# B&R Automation Studio project SCR
Automation Studio 4.0.18.71 SP

## Logical view

Binary libraries used (declarations not repeated): operator, runtime, astime, AsIecCon

### Global.var - Global variables
```iecst
(********************************************************************
 * COPYRIGHT --
 ********************************************************************
 * File: Global.var
 * Author: Arkadiusz
 * Created: April 16, 2018
 ********************************************************************
 * Global variables of project test2
 ********************************************************************)
VAR
	zadajnik : USINT;
	output2 : USINT;
	output1 : USINT;
	input3 : USINT;
	input2 : USINT;
	input1 : USINT;
	subs2Value : USINT;
	subs1Value : USINT;
	valuesSetFlag : USINT := 0;
END_VAR
```


### Program Logical/NastawaPWM (ANSIC) - Program

#### NastawaPWMCyclic.c - Cyclic code
```c
/********************************************************************
 * COPYRIGHT --
 ********************************************************************
 * Program: NastawaPWM
 * File: NastawaPWMCyclic.c
 * Author: Arkadiusz
 * Created: April 23, 2018
 ********************************************************************
 * Implementation of program NastawaPWM
 ********************************************************************/

#include <bur/plctypes.h>

#ifdef _DEFAULT_INCLUDES
	#include <AsDefault.h>
#endif

void _CYCLIC NastawaPWMCyclic(void)
{
	const double mnoznik = 0.027;
	wynikNastawy = inputAnalogowy * mnoznik;

	inputPerc = wynikNastawy;
	inputT_Ms = 20000;
	const cycleTime = 10;
	cycleIterator = cycleIterator + 1;
	time = cycleIterator * cycleTime;
	upTime = ((double)inputPerc/100) * inputT_Ms;

	if (time < upTime)
	{
		out1 = 1;
	}
	else
	{
		out1 = 0;
	}

	if (time >= inputT_Ms)
	{
		time = 0;
		cycleIterator = 0;
	}
}
```

#### NastawaPWMInit.c - Initialization code
```c
/********************************************************************
 * COPYRIGHT --
 ********************************************************************
 * Program: NastawaPWM
 * File: NastawaPWMInit.c
 * Author: Arkadiusz
 * Created: April 23, 2018
 ********************************************************************
 * Implementation of program NastawaPWM
 ********************************************************************/

#include <bur/plctypes.h>

#ifdef _DEFAULT_INCLUDES
	#include <AsDefault.h>
#endif

void _INIT NastawaPWMInit(void)
{
	/* TODO: Add code here */
}
```

#### NastawaPWM.var - Local variables
```iecst
(********************************************************************
 * COPYRIGHT --
 ********************************************************************
 * Program: NastawaPWM
 * File: NastawaPWM.var
 * Author: Arkadiusz
 * Created: April 23, 2018
 ********************************************************************
 * Local variables of program NastawaPWM
 ********************************************************************)
VAR
	upTime : REAL;
	time : LREAL;
	inputPerc : USINT := 0;
	out1 : USINT := 0;
	cycleIterator : INT := 0;
	inputT_Ms : UDINT := 0;
	inputAnalogowy : INT;
	wynikNastawy : USINT;
	inputVolt : REAL;
END_VAR
```

### Program Logical/PWM (ANSIC) - Program

#### PWMCyclic.c - Cyclic code
```c
/********************************************************************
 * COPYRIGHT --
 ********************************************************************
 * Program: Testowy
 * File: TestowyCyclic.c
 * Author: Arkadiusz
 * Created: April 16, 2018
 ********************************************************************
 * Implementation of program Testowy
 ********************************************************************/

#include <bur/plctypes.h>

#ifdef _DEFAULT_INCLUDES
	#include <AsDefault.h>
#endif

void _CYCLIC TestowyCyclic(void)
{
	inputPerc = 50;
	inputT_Ms = 20000;
	const cycleTime = 10;
	cycleIterator = cycleIterator + 1;
	time = cycleIterator * cycleTime;
	upTime = ((double)inputPerc/100) * inputT_Ms;

	if (time < upTime)
	{
		out1 = 1;
	}
	else
	{
		out1 = 0;
	}

	if (time >= inputT_Ms)
	{
		time = 0;
		cycleIterator = 0;
	}

}
```

#### PWMInit.c - Initialization code
```c
/********************************************************************
 * COPYRIGHT --
 ********************************************************************
 * Program: Testowy
 * File: TestowyInit.c
 * Author: Arkadiusz
 * Created: April 16, 2018
 ********************************************************************
 * Implementation of program Testowy
 ********************************************************************/

#include <bur/plctypes.h>

#ifdef _DEFAULT_INCLUDES
	#include <AsDefault.h>
#endif

void _INIT TestowyInit(void)
{
	out1 = 0;

}
```

#### PWM.var - Local variables
```iecst
(********************************************************************
 * COPYRIGHT --
 ********************************************************************
 * Program: Testowy
 * File: Testowy.var
 * Author: Arkadiusz
 * Created: April 16, 2018
 ********************************************************************
 * Local variables of program Testowy
 ********************************************************************)
VAR
	upTime : REAL;
	time : LREAL;
	inputPerc : USINT := 0;
	out1 : USINT := 0;
	cycleIterator : INT := 0;
	inputT_Ms : UDINT := 0;
END_VAR
```

### Program Logical/Nastawa (ANSIC) - nastawaProgram

#### NastawaCyclic.c - Cyclic code
```c
/********************************************************************
 * COPYRIGHT --
 ********************************************************************
 * Program: Nastawa
 * File: NastawaCyclic.c
 * Author: Arkadiusz
 * Created: April 23, 2018
 ********************************************************************
 * Implementation of program Nastawa
 ********************************************************************/

#include <bur/plctypes.h>

#ifdef _DEFAULT_INCLUDES
	#include <AsDefault.h>
#endif

void _CYCLIC NastawaCyclic(void)
{
	const double mnoznik = 100.0/32768;
	wynikNastawy = (int) ( ( (double) inputAnalogowy ) * mnoznik);
	zadajnik = wynikNastawy;

}
```

#### NastawaInit.c - Initialization code
```c
/********************************************************************
 * COPYRIGHT --
 ********************************************************************
 * Program: Nastawa
 * File: NastawaInit.c
 * Author: Arkadiusz
 * Created: April 23, 2018
 ********************************************************************
 * Implementation of program Nastawa
 ********************************************************************/

#include <bur/plctypes.h>

#ifdef _DEFAULT_INCLUDES
	#include <AsDefault.h>
#endif

void _INIT NastawaInit(void)
{
	/* TODO: Add code here */
}
```

#### Nastawa.var - Local variables
```iecst
(********************************************************************
 * COPYRIGHT --
 ********************************************************************
 * Program: Nastawa
 * File: Nastawa.var
 * Author: Arkadiusz
 * Created: April 23, 2018
 ********************************************************************
 * Local variables of program Nastawa
 ********************************************************************)
VAR
	inputAnalogowy : INT;
	wynikNastawy : USINT;
END_VAR
```

### Program Logical/GettingInput (ANSIC) - Program

#### GettingInputCyclic.c - Cyclic code
```c
/********************************************************************
 * COPYRIGHT --
 ********************************************************************
 * Program: GettingInput
 * File: GettingInputCyclic.c
 * Author: Arkadiusz
 * Created: April 25, 2018
 ********************************************************************
 * Implementation of program GettingInput
 ********************************************************************/

#include <bur/plctypes.h>

#ifdef _DEFAULT_INCLUDES
	#include <AsDefault.h>
#endif

void _CYCLIC GettingInputCyclic(void)
{
	if (input1 == 1 && inputIterator == 0)
	{
		previousP1 = 1;
	}

	if (input1 == 0 && previousP1 == 1 )
	{
	 	subs1Value = zadajnik;
		inputIterator++;
		previousP1 = 0;
	}

	if (input1== 1 && inputIterator == 1)
	{
		previousP2 = 1;
	}

	if (input1 == 0 && previousP2 == 1 )
	{
		subs2Value = zadajnik;
		inputIterator--;
		previousP2 = 0;
	}
}
```

#### GettingInputInit.c - Initialization code
```c
/********************************************************************
 * COPYRIGHT --
 ********************************************************************
 * Program: GettingInput
 * File: GettingInputInit.c
 * Author: Arkadiusz
 * Created: April 25, 2018
 ********************************************************************
 * Implementation of program GettingInput
 ********************************************************************/

#include <bur/plctypes.h>

#ifdef _DEFAULT_INCLUDES
	#include <AsDefault.h>
#endif

void _INIT GettingInputInit(void)
{
	/* TODO: Add code here */
}
```

#### GettingInput.var - Local variables
```iecst
(********************************************************************
 * COPYRIGHT --
 ********************************************************************
 * Program: GettingInput
 * File: GettingInput.var
 * Author: Arkadiusz
 * Created: April 25, 2018
 ********************************************************************
 * Local variables of program GettingInput
 ********************************************************************)
VAR
	inputIterator : USINT := 0;
	previousP2 : USINT := 0;
	previousP1 : USINT := 0;
END_VAR
```
